KUKA KRL data list: PrepareMillingTools.dat

&ACCESS RVO1
DEFDAT PrepareMillingTools

   ENUM E_PrepProfileType FrameUpper,FrameHinge,FrameLock,FrameThreshold, LeafUpper,LeafBottom,LeafHinge,LeafLock

ENDDAT
